{attribute addProperty BoxType "EL6001--0000"}
{attribute addProperty Id "InputsAT %I*Inputs_DD54DA92192240OutputsAT %Q*Outputs_377610EF192240WcStateAT %I*WcState_F855686C1620InfoDataAT %I*InfoData_BC63D37F80100"}
{attribute addProperty CRC "3007837535"}
{attribute addProperty SizeInBites "480"}
{attribute addProperty SizeInBytes "60"}
TYPE EL6001_A7B322AF :
STRUCT
	{attribute addProperty Name "Inputs"}
	Inputs : Inputs_DD54DA92;
	{attribute addProperty Name "Outputs"}
	Outputs : Outputs_377610EF;
	{attribute addProperty Name "WcState"}
	WcState : WcState_F855686C;
	{attribute addProperty Name "InfoData"}
	InfoData : InfoData_BC63D37F;
END_STRUCT
END_TYPE

(* stored: Version 1.2.0.0, ProductVersion 3.1.4024.9
   DUT EL6001_A7B322AF: Id {6f801cea-194c-40ce-865f-88b5f88d4d86} *)
